// TIA Portal project "Prova_PLC" (V16)

(* hardware
DEVICE "S7-1200 station_1"  S7-1200 Station
   slot 0: "Telaio di montaggio_0"  S7-1200 Rack  Rack  V1.0
   slot 1: "PLC_1"  CPU 1211C DC/DC/DC  6ES7 211-1AE40-0XB0  V4.4
*)

// ===== PLC "PLC_1"  CPU 1211C DC/DC/DC =====

VAR_GLOBAL   // PLC tag table "Tabella delle variabili standard"
   "System_Byte" AT %MB1 : Byte;
   "FirstScan" AT %M1.0 : Bool;
   "DiagStatusUpdate" AT %M1.1 : Bool;
   "AlwaysTRUE" AT %M1.2 : Bool;
   "AlwaysFALSE" AT %M1.3 : Bool;
   "Clock_Byte" AT %MB0 : Byte;
   "Clock_10Hz" AT %M0.0 : Bool;
   "Clock_5Hz" AT %M0.1 : Bool;
   "Clock_2.5Hz" AT %M0.2 : Bool;
   "Clock_2Hz" AT %M0.3 : Bool;
   "Clock_1.25Hz" AT %M0.4 : Bool;
   "Clock_1Hz" AT %M0.5 : Bool;
   "Clock_0.625Hz" AT %M0.6 : Bool;
   "Clock_0.5Hz" AT %M0.7 : Bool;
   "man_auto" AT %I0.0 : Bool;
   "pulsante_1" AT %I0.1 : Bool;
   "pulsante_2" AT %I0.2 : Bool;
   "emergenza" AT %I0.3 : Bool;
   "pulsante_3" AT %I0.4 : Bool;
   "luce_1" AT %Q0.0 : Bool;
   "luce_2" AT %Q0.1 : Bool;
   "sensoreProssimita" AT %I0.5 : Bool;
END_VAR

DATA_BLOCK "DB_dati"   // DB1
{ S7_Optimized_Access := 'TRUE' }
VERSION : 0.1
   VAR
      memoria : Bool;
      cnt : Int;
   END_VAR
BEGIN
END_DATA_BLOCK

// folder: System blocks/Program resources

DATA_BLOCK "IEC_Counter_0_DB"   // DB2
{ S7_Optimized_Access := 'TRUE' }
AUTHOR : Simatic
FAMILY : IEC
NAME : CNTR
VERSION : 1.0
// stored: InstanceOfName IEC_COUNTER
"IEC_COUNTER"
BEGIN
END_DATA_BLOCK

// folder: (top level)

FUNCTION "contatore" : Void   // FC1, LAD
{ S7_Optimized_Access := 'TRUE' }
VERSION : 0.1
BEGIN

REGION Network 1
   // premo luce2, inizia a lampeggiare uscita luce1; quando sensore prossimita conta 10 passaggi, si accende la luce1 e si spegna la luce1; con il tast luce2 si resetta lo stato, lasciando acceso però la luce1 fissa; quando ripremo lo start (pulsante luce2), la luce1 inizia a lampeggiare.
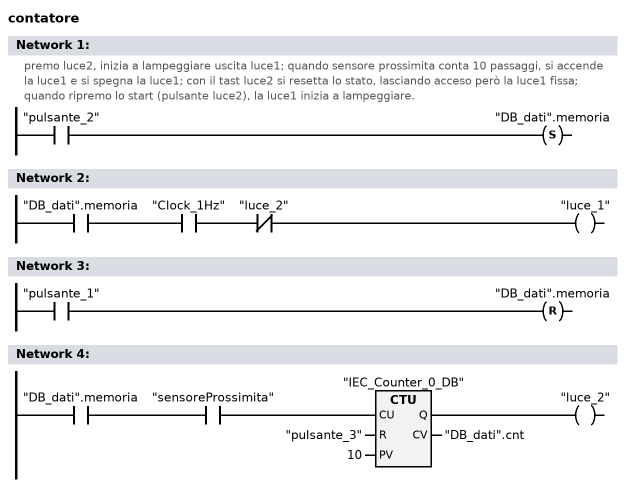
   RUNG wire#powerrail
      Contact( "pulsante_2" )
      S_Coil( "DB_dati".memoria )
   END_RUNG
   // the same network as SCL:
   IF "pulsante_2" THEN "DB_dati".memoria := TRUE; END_IF;
END_REGION

REGION Network 2
   RUNG wire#powerrail
      Contact( "DB_dati".memoria )
      Contact( "Clock_1Hz" )
      I_Contact( "luce_2" )
      Coil( "luce_1" )
   END_RUNG
   // the same network as SCL:
   "luce_1" := "DB_dati".memoria AND "Clock_1Hz" AND NOT "luce_2";
END_REGION

REGION Network 3
   RUNG wire#powerrail
      Contact( "pulsante_1" )
      R_Coil( "DB_dati".memoria )
   END_RUNG
   // the same network as SCL:
   IF "pulsante_1" THEN "DB_dati".memoria := FALSE; END_IF;
END_REGION

REGION Network 4
   "IEC_Counter_0_DB".CTU(CU := "DB_dati".memoria AND "sensoreProssimita",
                          R := "pulsante_3",
                          PV := 10,
                          CV => "DB_dati".cnt);
   "luce_2" := "IEC_Counter_0_DB".Q;
END_REGION
END_FUNCTION

ORGANIZATION_BLOCK "Main"   // OB1, LAD, ProgramCycle
TITLE = "Main Program Sweep (Cycle)"
{ S7_Optimized_Access := 'TRUE' }
VERSION : 0.1
   VAR_INPUT
      Initial_Call : Bool;   // Initial call of this OB
      Remanence : Bool;   // =True, if remanent data are available
   END_VAR
BEGIN

REGION Network 1
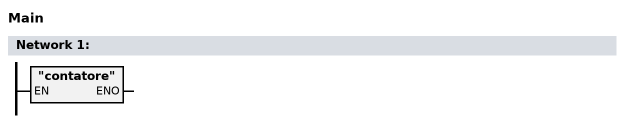
   RUNG wire#powerrail
      "contatore"()
   END_RUNG
   // the same network as SCL:
   "contatore"();
END_REGION
END_ORGANIZATION_BLOCK